Universal Robots URScript: execute_drop_action.script

def execute_drop_action():
    target_pose = pose_add(get_actual_tcp_pose(), p[0, 0, -0.1, 0, 0, 0])
    movel(target_pose)
    set_standard_digital_out(0, False)
end
